# EPICS autosave request: iocBoot/iocSimEpics/auto_settings.req
file "simEpics.req", P=$(P), R=$(R)
file "simEpics_settings.req", P=$(P), R=$(R)
